PROGRAM P_Strategy
VAR
	fbSensor1		: FB_PT100;
	fbMotor1		: FB_Motor_PT(TempSensor := fbSensor1);
	fbSensor2		: FB_PT1000;
	fbMotor2		: FB_Motor_PT(fbSensor2);
END_VAR

// Motors
fbSensor1();
fbMotor1();	
fbSensor2();
fbMotor2();

END_PROGRAM

(* stored: Version 1.1.0.1, ProductVersion 3.1.4024.12
   POU P_Strategy: Id {71eab6f8-9f1c-4cb6-8e46-fa257ca9189d}, SpecialFunc None *)
